FUNCTION_BLOCK container_one
  (* Standard: 61499-2 *)
  (* Version 0.1, 2017-00-09, Hammond, HAMMONDSDESKTOP *)
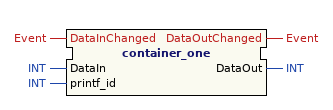
  EVENT_INPUT
    DataInChanged;
  END_EVENT
  EVENT_OUTPUT
    DataOutChanged;
  END_EVENT
  VAR_INPUT
    DataIn : INT;
    printf_id : INT;
  END_VAR
  VAR_OUTPUT
    DataOut : INT;
  END_VAR
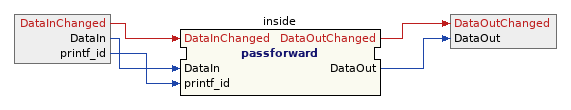
  FBS
    inside : passforward;
  END_FBS
  EVENT_CONNECTIONS
    DataInChanged TO inside.DataInChanged;
    inside.DataOutChanged TO DataOutChanged;
  END_CONNECTIONS
  DATA_CONNECTIONS
    DataIn TO inside.DataIn;
    printf_id TO inside.printf_id;
    inside.DataOut TO DataOut;
  END_CONNECTIONS
END_FUNCTION_BLOCK
